FUNCTION_BLOCK FB_Animal IMPLEMENTS I_Animal
VAR
	 sOutput : STRING := '';
END_VAR

METHOD M_Eat
THIS^.sOutput := 'Animal eats food';
END_METHOD

METHOD M_Sleep : BOOL
THIS^.sOutput := 'Animal sleeps';
END_METHOD

END_FUNCTION_BLOCK

(* stored: Version 1.1.0.1, ProductVersion 3.1.4024.16
   POU FB_Animal: Id {53f8f5ba-dd2e-4c6a-8f33-0eba62063c7e}, SpecialFunc None
   Method M_Eat: Id {17971ee3-69a1-47c4-b9d6-36a2ccfb1e14}
   Method M_Sleep: Id {8a1ed1d1-92cd-4b90-810f-c154f92c31a4} *)
